Omron CX-Programmer project NewProject (CX-Programmer 9.75)

# PLC NewPLC1: CJ2M CPU11

## Global symbols (name address type ; comment)
Always_ON 0.11 BOOL

## Program NewProgram1 (cyclic task 0)
Local symbols
ALM_E_Stop W200.06 BOOL
ALM_FD_Fan_OL W200.04 BOOL
ALM_Flame_Failure W200.02 BOOL
ALM_High_Temp W200.00 BOOL
ALM_ID_Fan_OL W200.03 BOOL
ALM_Kiln_Motor_OL W200.05 BOOL
ALM_Low_Pressure W200.01 BOOL
ALM_Sensor_Fault W200.07 BOOL
Alarm_Horn 100.06 BOOL
Auto_Enable W0.08 BOOL
Beacon_Light 100.07 BOOL
Burner_Ready 0.07 BOOL  ; Burner Ready
Conveyor_Run 100.05 BOOL
Critical_Fault W0.05 BOOL
E_Stop 0.02 BOOL  ; Emergency Stop
FD_Fan_FB 0.05 BOOL  ; FD Fan Feedback
FD_Fan_OL 0.09 BOOL  ; FD Fan Overload
FD_Fan_Run 100.01 BOOL
Flame_Detector 0.03 BOOL  ; Flame Scanner
Flame_Proven W0.03 BOOL
Fuel_Flow_PV D114 REAL
Fuel_Flow_Raw D102 UINT
Fuel_Valve_Open 100.03 BOOL
High_Temp 0.12 BOOL
ID_Fan_FB 0.04 BOOL  ; ID Fan Feedback
ID_Fan_OL 0.08 BOOL  ; ID Fan Overload
ID_Fan_Run 100.00 BOOL
Igniter_Run 100.04 BOOL
Kiln_Motor_FB 0.06 BOOL  ; Kiln Motor Feedback
Kiln_Motor_OL 0.10 BOOL  ; Kiln Motor Overload
Kiln_Motor_Run 100.02 BOOL
Kiln_Pressure_PV D112 REAL
Kiln_Temp_PV D110 REAL
Kiln_Temp_Raw D100 UINT
Kiln_Temp_SP D200 REAL
Manual_Mode W0.09 BOOL
Oxygen_PV D116 REAL
Oxygen_Raw D103 UINT
PID_Enable W0.07 BOOL
PID_Error D206 REAL
PID_Output D204 REAL
Permissive_OK W0.01 BOOL
Pressure_Raw D101 UINT
Purge_Complete W0.02 BOOL
Run_Command W0.00 BOOL
ST_ESTOP W100.08 BOOL
ST_EStop BOOL
ST_FAULT W100.09 BOOL
ST_FLAME_VERIFY W100.04 BOOL
ST_IDLE W100.00 BOOL
ST_IGNITION W100.03 BOOL
ST_PRESTART W100.01 BOOL
ST_PRODUCTION W100.06 BOOL
ST_PURGE W100.02 BOOL
ST_SHUTDOWN W100.07 BOOL
ST_WARMUP W100.05 BOOL
Shutdown_Request W0.06 BOOL
Start_PB 0.00 BOOL  ; Start Pushbutton
Stop_PB 0.01 BOOL  ; Stop Pushbutton
Temp_Ready W0.04 BOOL

### Section Section1

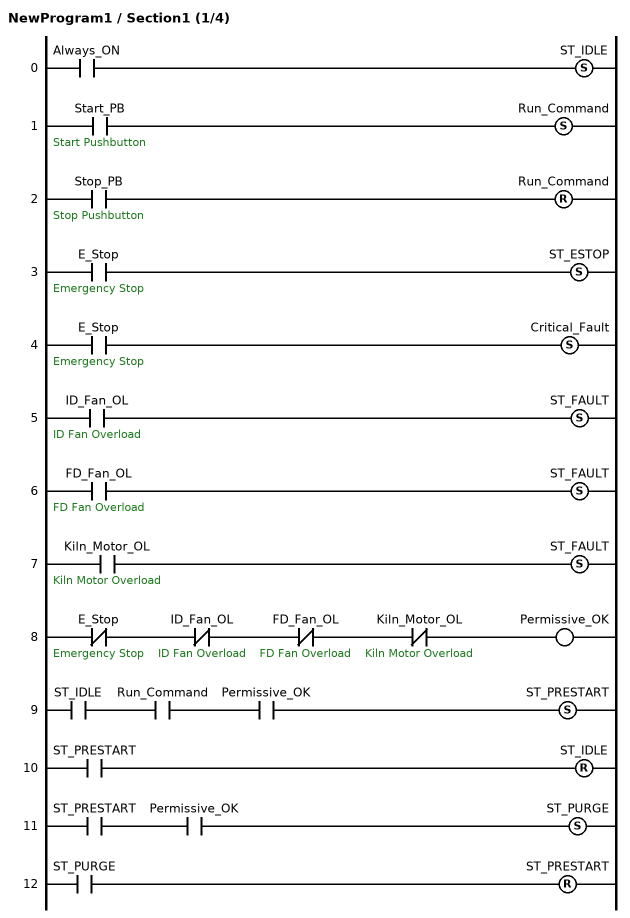
; rung 0
LD Always_ON
SET ST_IDLE
; rung 1
LD Start_PB  ; Start Pushbutton
SET Run_Command
; rung 2
LD Stop_PB  ; Stop Pushbutton
RSET Run_Command
; rung 3
LD E_Stop  ; Emergency Stop
SET ST_ESTOP
; rung 4
LD E_Stop  ; Emergency Stop
SET Critical_Fault
; rung 5
LD ID_Fan_OL  ; ID Fan Overload
SET ST_FAULT
; rung 6
LD FD_Fan_OL  ; FD Fan Overload
SET ST_FAULT
; rung 7
LD Kiln_Motor_OL  ; Kiln Motor Overload
SET ST_FAULT
; rung 8
LDNOT E_Stop  ; Emergency Stop
ANDNOT ID_Fan_OL  ; ID Fan Overload
ANDNOT FD_Fan_OL  ; FD Fan Overload
ANDNOT Kiln_Motor_OL  ; Kiln Motor Overload
OUT Permissive_OK
; rung 9
LD ST_IDLE
AND Run_Command
AND Permissive_OK
SET ST_PRESTART
; rung 10
LD ST_PRESTART
RSET ST_IDLE
; rung 11
LD ST_PRESTART
AND Permissive_OK
SET ST_PURGE
; rung 12
LD ST_PURGE
RSET ST_PRESTART

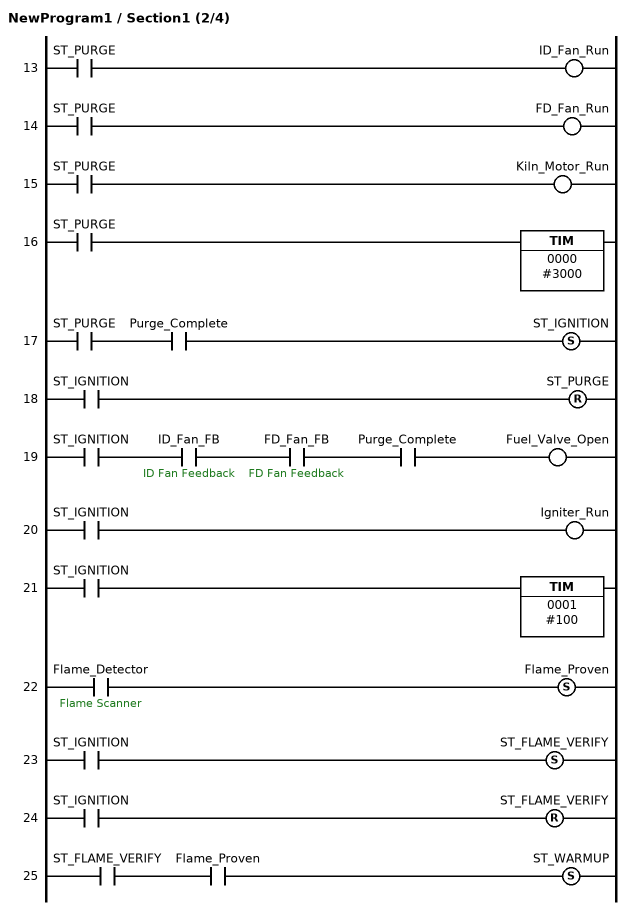
; rung 13
LD ST_PURGE
OUT ID_Fan_Run
; rung 14
LD ST_PURGE
OUT FD_Fan_Run
; rung 15
LD ST_PURGE
OUT Kiln_Motor_Run
; rung 16
LD ST_PURGE
TIM 0000 #3000
; rung 17
LD ST_PURGE
AND Purge_Complete
SET ST_IGNITION
; rung 18
LD ST_IGNITION
RSET ST_PURGE
; rung 19
LD ST_IGNITION
AND ID_Fan_FB  ; ID Fan Feedback
AND FD_Fan_FB  ; FD Fan Feedback
AND Purge_Complete
OUT Fuel_Valve_Open
; rung 20
LD ST_IGNITION
OUT Igniter_Run
; rung 21
LD ST_IGNITION
TIM 0001 #100
; rung 22
LD Flame_Detector  ; Flame Scanner
SET Flame_Proven
; rung 23
LD ST_IGNITION
SET ST_FLAME_VERIFY
; rung 24
LD ST_IGNITION
RSET ST_FLAME_VERIFY
; rung 25
LD ST_FLAME_VERIFY
AND Flame_Proven
SET ST_WARMUP

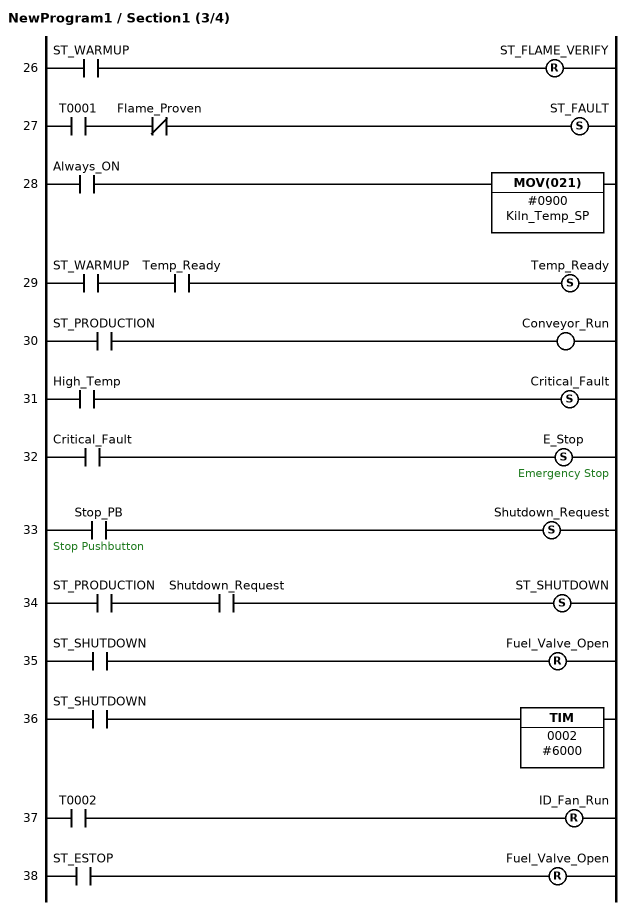
; rung 26
LD ST_WARMUP
RSET ST_FLAME_VERIFY
; rung 27
LD T0001
ANDNOT Flame_Proven
SET ST_FAULT
; rung 28
LD Always_ON
MOV(021) #0900 Kiln_Temp_SP
; rung 29
LD ST_WARMUP
AND Temp_Ready
SET Temp_Ready
; rung 30
LD ST_PRODUCTION
OUT Conveyor_Run
; rung 31
LD High_Temp
SET Critical_Fault
; rung 32
LD Critical_Fault
SET E_Stop  ; Emergency Stop
; rung 33
LD Stop_PB  ; Stop Pushbutton
SET Shutdown_Request
; rung 34
LD ST_PRODUCTION
AND Shutdown_Request
SET ST_SHUTDOWN
; rung 35
LD ST_SHUTDOWN
RSET Fuel_Valve_Open
; rung 36
LD ST_SHUTDOWN
TIM 0002 #6000
; rung 37
LD T0002
RSET ID_Fan_Run
; rung 38
LD ST_ESTOP
RSET Fuel_Valve_Open

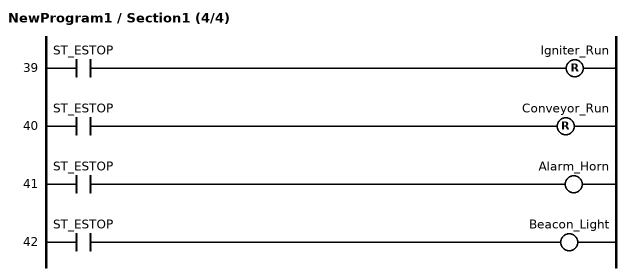
; rung 39
LD ST_ESTOP
RSET Igniter_Run
; rung 40
LD ST_ESTOP
RSET Conveyor_Run
; rung 41
LD ST_ESTOP
OUT Alarm_Horn
; rung 42
LD ST_ESTOP
OUT Beacon_Light

### Section END
; rung 0
END(001)